{attribute 'qualified_only'}
{attribute 'strict'}
{attribute 'to_string'}
TYPE E_EcState1 :
(
	enum_member := 0
);
END_TYPE

(* stored: Version 1.1.0.1, ProductVersion 3.1.4026.8
   DUT E_EcState1: Id {4e51b496-c495-4359-bb9c-7b8cf6125391} *)
